% RSLogix 500 project pulse_rotameter.RSS, saved by version 8.30.00.16 %
PROJECT "UNTITLED"    % processor: Bul.1763 MicroLogix 1100 Series B %

PROGRAM FILES
  LAD 2 "MAIN"  2 rungs
  LAD 3 "INPUT"  1 rungs
  LAD 4 "OUTPUT"  1 rungs
  LAD 5 "CONTROL"  7 rungs

DATA FILES
  O0 OUTPUT  4 elements
  I1 INPUT  6 elements
  S2 STATUS  66 elements
  B3 BINARY  2 elements
  T4 TIMER  2 elements
  C5 COUNTER  1 elements
  R6 CONTROL  1 elements
  N7 INTEGER  1 elements
  F8 FLOAT  2 elements

LADDER 2 "MAIN"
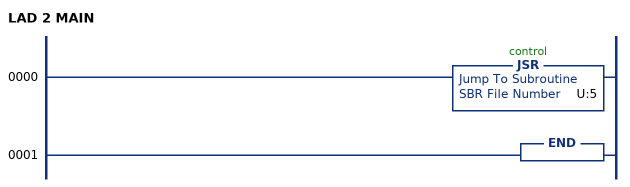
% Rung: 0 %
SOR JSR U:5 EOR
%   U:5  "control" %
% Rung: 1 %
SOR END EOR

LADDER 5 "CONTROL"
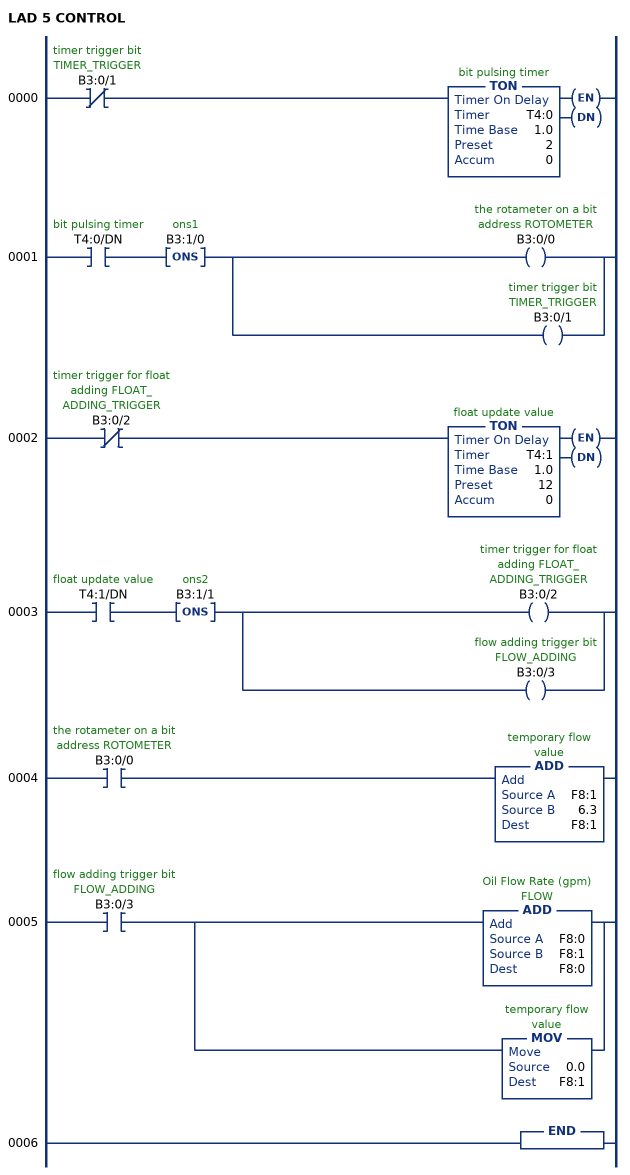
% Rung: 0 %
SOR XIO B3:0/1 TON T4:0 1.0 2 0 EOR
%   B3:0/1  TIMER_TRIGGER  "timer trigger bit" %
%   T4:0  "bit pulsing timer" %
% Rung: 1 %
SOR XIC T4:0/DN ONS B3:1/0 BST OTE B3:0/0 NXB OTE B3:0/1 BND EOR
%   T4:0  "bit pulsing timer" %
%   B3:1/0  "ons1" %
%   B3:0/0  ROTOMETER  "the rotameter on a bit address" %
%   B3:0/1  TIMER_TRIGGER  "timer trigger bit" %
% Rung: 2 %
SOR XIO B3:0/2 TON T4:1 1.0 12 0 EOR
%   B3:0/2  FLOAT_ADDING_TRIGGER  "timer trigger for float adding" %
%   T4:1  "float update value" %
% Rung: 3 %
SOR XIC T4:1/DN ONS B3:1/1 BST OTE B3:0/2 NXB OTE B3:0/3 BND EOR
%   T4:1  "float update value" %
%   B3:1/1  "ons2" %
%   B3:0/2  FLOAT_ADDING_TRIGGER  "timer trigger for float adding" %
%   B3:0/3  FLOW_ADDING  "flow adding trigger bit" %
% Rung: 4 %
SOR XIC B3:0/0 ADD F8:1 6.3 F8:1 EOR
%   B3:0/0  ROTOMETER  "the rotameter on a bit address" %
%   F8:1  "temporary flow value" %
% Rung: 5 %
SOR XIC B3:0/3 BST ADD F8:0 F8:1 F8:0 NXB MOV 0.0 F8:1 BND EOR
%   B3:0/3  FLOW_ADDING  "flow adding trigger bit" %
%   F8:0  FLOW  "Oil Flow Rate (gpm)" %
%   F8:1  "temporary flow value" %
% Rung: 6 %
SOR END EOR

DATA TABLE (non-zero values as saved)
DATA T4
% .PRE .ACC %
% T4:0 % 2 0
% T4:1 % 12 0
